{attribute 'GeneratedUsingTerminal: AT2000-0233-0022'}
{attribute addProperty BoxType "AT2000-0233-0022"}
{attribute addProperty Id "StatusAT %I*UINT2Current_actual_value_ChAT %I*ARRAY[0..13] OF INT28"}
{attribute addProperty CRC "3830004940"}
{attribute addProperty Size "30"}
TYPE CC_Inputs_14_Ch_F1B79554 :
STRUCT
	{attribute addProperty Name "Status"}
	Status AT %I* : UINT;
	{attribute addProperty Name "Current_actual_value_Ch"}
	Current_actual_value_Ch AT %I* : ARRAY[0..13] OF INT;
END_STRUCT
END_TYPE

(* stored: Version 1.2.0.0, ProductVersion 3.1.4024.9
   DUT CC_Inputs_14_Ch_F1B79554: Id {f57af807-edc5-424c-9636-1f569001cb08} *)
